# EPICS substitutions: modules/event/evrSupport/Db/ioc/IOC-IN20-LS19evr.substitutions
#==============================================================================
#
# Abs:  LCLS EVR IOC records for IN20 LS19
#
# Name: IOC-IN20-LS19evr.substitutions
#
#==============================================================================
#
file evrLSXX.db
{
pattern { DEVICE        }
	{ EVR:IN20:LS19 }
}
